TYPE AT_FloorCalls1 : ARRAY[0..50] OF ST_FloorCall;
END_TYPE

(* stored: Version 1.1.0.1, ProductVersion 3.1.4024.16
   DUT AT_FloorCalls1: Id {8091e8de-a29b-493a-80c5-a0923562787a} *)
